TYPE ST_Shelf :
STRUCT
	nPosition 	: DINT;
	bConfigured : BOOL;
END_STRUCT
END_TYPE

(* stored: Version 1.1.0.1, ProductVersion 3.1.4024.11
   DUT ST_Shelf: Id {9af2295b-d1e4-444a-895a-1c614985a9ef} *)
